FUNCTION_BLOCK DigitalInput IMPLEMENTS I_DigitalInput
VAR_INPUT
END_VAR
VAR_OUTPUT
END_VAR
VAR
	ID:				STRING(25);
	Input			AT%I*: BOOL;
END_VAR

METHOD FB_init : BOOL
VAR_INPUT
	bInitRetains : BOOL; // if TRUE, the retain variables are initialized (warm start / cold start)
	bInCopyCode : BOOL;  // if TRUE, the instance afterwards gets moved into the copy code (online change)
	ID:			String(25);
END_VAR
this^.ID:= ID;
END_METHOD

PROPERTY PUBLIC P_ID : String(25)
GET
P_ID:= ID;
END_GET
END_PROPERTY

PROPERTY PUBLIC P_Value : bool
GET
P_Value:= Input;
END_GET
END_PROPERTY

END_FUNCTION_BLOCK

(* stored: Version 1.1.0.1
   POU DigitalInput: Id {8904ca26-c33a-0d5e-01bd-927c832f4cd0}, SpecialFunc None
   Method FB_init: Id {bc5bb0ce-93c3-0bde-1d49-3a327da4d83a}
   Property P_ID: Id {d2592e33-0c09-00ed-2a19-2a2ac1387854}
   Get Get: Id {db03f916-1db4-0ef0-2610-a102e9e38d81}
   Property P_Value: Id {eb10c2b4-f572-0e2d-2bec-edb3aca0020c}
   Get Get: Id {0af5f71f-a62f-0bc9-1f1b-442ea0defb72} *)
